// TIA Portal V18 export
FUNCTION "Output" : Void   // FC32, LAD
{ S7_Optimized_Access := 'TRUE' }
VERSION : 0.1
// stored: AutoNumber true, IsIECCheckEnabled false, SetENOAutomatically false, UDAEnableTagReadback false
BEGIN

REGION Network 1: tower lamp amber
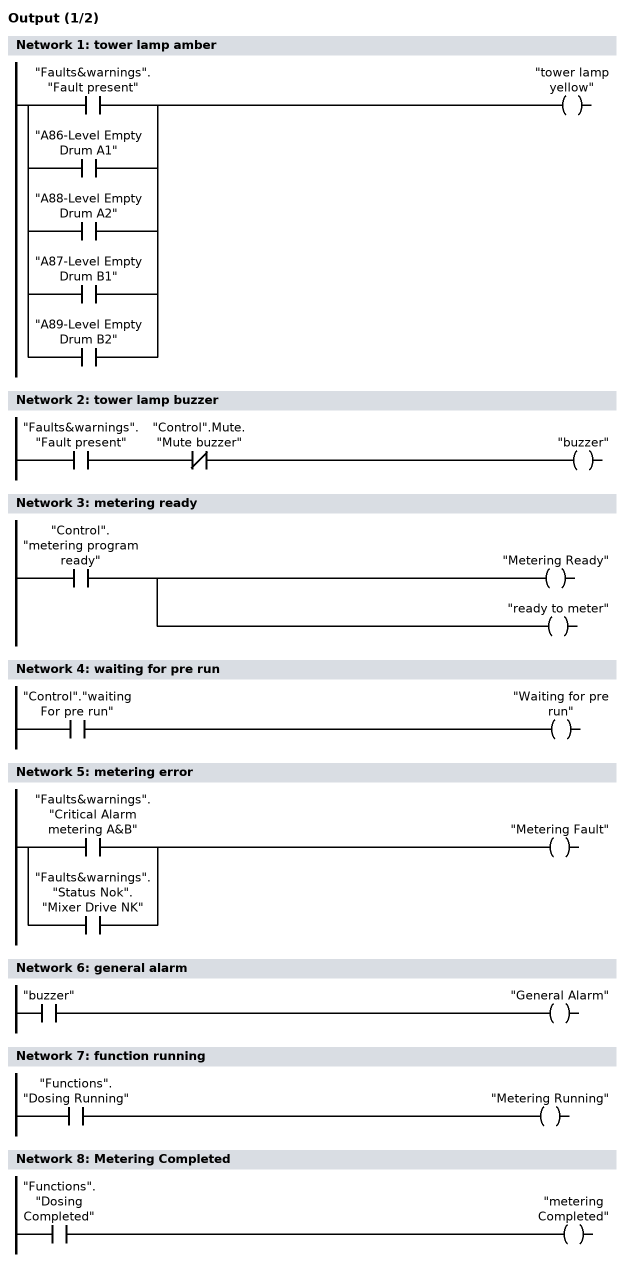
   RUNG wire#powerrail
      Contact( "Faults&warnings"."Fault present" )
      wire#w1
      Coil( "tower lamp yellow" )
   END_RUNG
   RUNG wire#powerrail
      Contact( "A86-Level Empty Drum A1" )
   END_RUNG wire#w1
   RUNG wire#powerrail
      Contact( "A88-Level Empty Drum A2" )
   END_RUNG wire#w1
   RUNG wire#powerrail
      Contact( "A87-Level Empty Drum B1" )
   END_RUNG wire#w1
   RUNG wire#powerrail
      Contact( "A89-Level Empty Drum B2" )
   END_RUNG wire#w1
   // the same network as SCL:
   "tower lamp yellow" := "Faults&warnings"."Fault present" OR "A86-Level Empty Drum A1" OR "A88-Level Empty Drum A2" OR "A87-Level Empty Drum B1" OR "A89-Level Empty Drum B2";
END_REGION

REGION Network 2: tower lamp buzzer
   RUNG wire#powerrail
      Contact( "Faults&warnings"."Fault present" )
      I_Contact( "Control".Mute."Mute buzzer" )
      Coil( "buzzer" )
   END_RUNG
   // the same network as SCL:
   "buzzer" := "Faults&warnings"."Fault present" AND NOT "Control".Mute."Mute buzzer";
END_REGION

REGION Network 3: metering ready
   RUNG wire#powerrail
      Contact( "Control"."metering program ready" )
      wire#w1
      Coil( "Metering Ready" )
   END_RUNG
   RUNG wire#w1
      Coil( "ready to meter" )
   END_RUNG
   // the same network as SCL:
   "Metering Ready" := "Control"."metering program ready";
   "ready to meter" := "Control"."metering program ready";
END_REGION

REGION Network 4: waiting for pre run
   RUNG wire#powerrail
      Contact( "Control"."waiting For pre run" )
      Coil( "Waiting for pre run" )
   END_RUNG
   // the same network as SCL:
   "Waiting for pre run" := "Control"."waiting For pre run";
END_REGION

REGION Network 5: metering error
   RUNG wire#powerrail
      Contact( "Faults&warnings"."Critical Alarm metering A&B" )
      wire#w1
      Coil( "Metering Fault" )
   END_RUNG
   RUNG wire#powerrail
      Contact( "Faults&warnings"."Status Nok"."Mixer Drive NK" )
   END_RUNG wire#w1
   // the same network as SCL:
   "Metering Fault" := "Faults&warnings"."Critical Alarm metering A&B" OR "Faults&warnings"."Status Nok"."Mixer Drive NK";
END_REGION

REGION Network 6: general alarm
   RUNG wire#powerrail
      Contact( "buzzer" )
      Coil( "General Alarm" )
   END_RUNG
   // the same network as SCL:
   "General Alarm" := "buzzer";
END_REGION

REGION Network 7: function running
   RUNG wire#powerrail
      Contact( "Functions"."Dosing Running" )
      Coil( "Metering Running" )
   END_RUNG
   // the same network as SCL:
   "Metering Running" := "Functions"."Dosing Running";
END_REGION

REGION Network 8: Metering Completed
   RUNG wire#powerrail
      Contact( "Functions"."Dosing Completed" )
      Coil( "metering Completed" )
   END_RUNG
   // the same network as SCL:
   "metering Completed" := "Functions"."Dosing Completed";
END_REGION

REGION Network 9: Control On Lamp
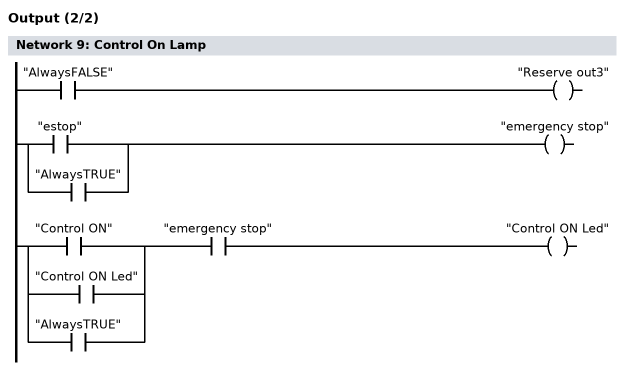
   RUNG wire#powerrail
      Contact( "AlwaysFALSE" )
      Coil( "Reserve out3" )
   END_RUNG
   RUNG wire#powerrail
      Contact( "estop" )
      wire#w1
      Coil( "emergency stop" )
   END_RUNG
   RUNG wire#powerrail
      Contact( "AlwaysTRUE" )
   END_RUNG wire#w1
   RUNG wire#powerrail
      Contact( "Control ON" )
      wire#w2
      Contact( "emergency stop" )
      Coil( "Control ON Led" )
   END_RUNG
   RUNG wire#powerrail
      Contact( "Control ON Led" )
   END_RUNG wire#w2
   RUNG wire#powerrail
      Contact( "AlwaysTRUE" )
   END_RUNG wire#w2
   // the same network as SCL:
   "Reserve out3" := "AlwaysFALSE";
   "emergency stop" := "estop" OR "AlwaysTRUE";
   "Control ON Led" := ("Control ON" OR "Control ON Led" OR "AlwaysTRUE") AND "emergency stop";
END_REGION
END_FUNCTION
